FUNCTION_BLOCK W3W1
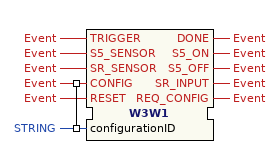
  EVENT_INPUT
    TRIGGER;
    S5_SENSOR;
    SR_SENSOR;
    CONFIG WITH configurationID;
    RESET;
  END_EVENT
  EVENT_OUTPUT
    DONE;
    S5_ON;
    S5_OFF;
    SR_INPUT;
    REQ_CONFIG;
  END_EVENT
  VAR_INPUT
    configurationID : STRING;
  END_VAR
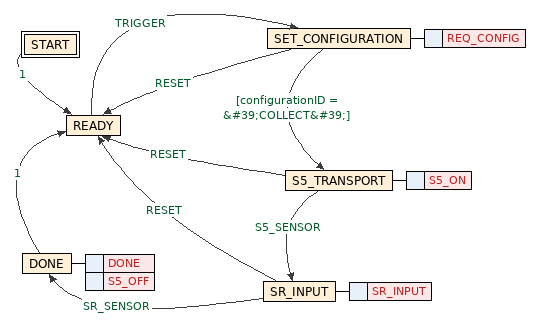
  EC_STATES
    START;
    SR_INPUT : -> SR_INPUT;
    S5_TRANSPORT : -> S5_ON;
    DONE : -> DONE, -> S5_OFF;
    READY;
    SET_CONFIGURATION : -> REQ_CONFIG;
  END_STATES
  EC_TRANSITIONS
    START TO READY := 1;
    SR_INPUT TO DONE := SR_SENSOR;
    READY TO SET_CONFIGURATION := TRIGGER;
    SET_CONFIGURATION TO S5_TRANSPORT := [configurationID = &#39;COLLECT&#39;];
    DONE TO READY := 1;
    S5_TRANSPORT TO SR_INPUT := S5_SENSOR;
    SET_CONFIGURATION TO READY := RESET;
    S5_TRANSPORT TO READY := RESET;
    SR_INPUT TO READY := RESET;
  END_TRANSITIONS
  ALGORITHM INIT IN ST:

  END_ALGORITHM
  ALGORITHM REQ IN ST:

  END_ALGORITHM
END_FUNCTION_BLOCK
